FUNCTION_BLOCK FB_MotorControl IMPLEMENTS I_MotorControl
VAR
	fbVfdIOControl: FB_VFDIOControl;
END_VAR

METHOD GetActualSpeed : INT
GetActualSpeed := fbVfdIOControl.nActualSpeed;
END_METHOD

PROPERTY RemoteLocalStatus : BOOL
GET
RemoteLocalStatus := fbVfdIOControl.bRemoteLocalStatus;
END_GET
END_PROPERTY

METHOD SetSpeed : BOOL
VAR_input
	nSetSpeed	: INT;
END_VAR
fbVfdIOControl.nSetSpeed := nSetSpeed;
END_METHOD

METHOD StartMotor : BOOL
VAR_INPUT
	bStart: BOOL;
END_VAR
fbVfdIOControl.bStartMotor := bStart;
END_METHOD

METHOD StopMotor : BOOL
VAR_INPUT
	bStop: BOOL;
END_VAR
fbVfdIOControl.bStopMotor := bStop;
END_METHOD

END_FUNCTION_BLOCK

(* stored: Version 1.1.0.1, ProductVersion 3.1.4024.4
   POU FB_MotorControl: Id {59012f19-5ded-477a-b381-91a15662779c}, SpecialFunc None
   Method GetActualSpeed: Id {81a8c47b-7b66-47f2-832d-a3855e9a9429}
   Property RemoteLocalStatus: Id {3f54db94-bbc1-4da1-86f8-27a87e796e7a}
   Get Get: Id {dd4c6e53-00ec-43fc-972e-b899817708fe}
   Method SetSpeed: Id {d5a6d8eb-b97f-405f-a579-2da1bb17ed85}
   Method StartMotor: Id {b058c898-eeb4-4dfd-8e11-01b32ed170cc}
   Method StopMotor: Id {fdb0a518-a5b6-4232-9f58-f57da886b15d} *)
